// TIA Portal V21 export
DATA_BLOCK "N2Sparging"   // DB307
AUTHOR : PRECISE
FAMILY : PRECISE
// stored: AutoNumber false, InstanceOfName FB303, InstanceOfType FB
"FB303"
   // VAR_INPUT
   //    Enable : Bool;
   //    Disable : Bool;
   //    Fault : Bool;
   //    SecPulse : Bool;
   //    AlwaysTrue { ExternalVisible := 'False'} : Bool;
   //    StartConfirmationPopupSel : Bool;
   //    EndConfirmationPopupSel : Bool;
   //    SpargingModeSel : Int := 1;
   //    SpargingTimebaseSel : Bool;
   //    SpargingLineSel : Bool;   // Sparging LineSelection: 0-THRU N2 FILTER /1-THRU VV
   //    GasSel : Int := 1;   // N2 Selection - 0-AIR/1-N2
   //    SetDO : Real := 10.2;
   //    SpargingTimeMin : Int := 2;
   //    SpargingTimeSec : Int := 0;
   //    PressuretoOpenVV : Real;
   //    PressuretoCloseVV : Real;
   //    ActualDO : Real;
   //    ActualPressure : Real;
   //    DelaytoOpenGasIn : Int;
   // END_VAR
   // VAR_OUTPUT
   //    AirValve : Bool;
   //    N2Valve : Bool;
   //    SpargingLineValves : Bool;
   //    VentValve : Bool;
   //    StartConfirmationPopup : Bool;
   //    EndConfirmationPopup : Bool;
   //    SpargingTimeMinPV : DInt;
   //    SpargingTimeSecPV : DInt;
   //    PrintTrigger { ExternalAccessible := 'False'; ExternalVisible := 'False'; ExternalWritable := 'False'} : Bool;
   //    PrintWord : Int;
   //    PrintStatus : String[50];
   // END_VAR
   // VAR_IN_OUT
   //    Start : Bool;
   //    Stop : Bool;
   //    Reset : Bool;
   //    StartConfirmationAck : Bool;
   //    EndConfirmationAck : Bool;
   //    SpareBtn1 : Bool;
   //    SpareBtn2 : Bool;
   //    SpareBtn3 : Bool;
   //    Running : Bool;
   //    Selected : Bool;
   //    Paused : Bool;
   //    StartConfirmationPopupTemp : Bool;
   //    EndConfirmationPopupTemp : Bool;
   //    SpargingStarted : Bool;
   //    SpargingOver : Bool;
   //    SpargingTimerRunning : Bool;
   // END_VAR
   // VAR
   //    ValveOnDelayPV : Int;
   //    ValveOffDelayPV : Int;
   //    PrintTriggerTemp : Bool;
   //    RE1 : Bool;
   //    RE2 : Bool;
   //    RE3 : Bool;
   //    RE4 : Bool;
   //    RE5 : Bool;
   //    RE6 : Bool;
   //    RE7 : Bool;
   //    SpargingTimer : "FB101";
   //    PrintTriggerResetTimer { S7_SetPoint := 'True'} : TON_TIME;
   //    BtnResetTimer { S7_SetPoint := 'True'} : TON_TIME;
   // END_VAR
BEGIN
END_DATA_BLOCK
